Staubli VAL3: lffxx.dtx

jointRx oo = {j3=90, j5=90}
mdesc mNomSpeed
pointRx point0 = {x=850, z=300, rx=-180, rz=-180, fatherId=world[0]}
tool tool1 = {z=94, fatherId=flange[0], ioLink=valve1}
